PROGRAM PRG_Parada
VAR
	EstoyBloqueandoA: BOOL;
	EstoyBloqueandoV: BOOL;
	EstoyBloqueandoM: BOOL;

	StopBladeA: FB_StopBlade;
	CintaA: 	FB_Cinta;
	
	StopBladeV: FB_StopBlade;
	CintaV: 	FB_Cinta;
	
	StopBladeM: FB_StopBlade;
	CintaM: 	FB_Cinta;
	
	bBloqueoPusherA: BOOL;
	bBloqueoPusherV: BOOL;
	bBloqueoPusherM: BOOL;
END_VAR

(* Mediante este POU se controla el apagado de las líneas en caso de que comiencen a entrar demasiadas piezas en una misma
línea. Mediante su llamada, se impide que haya más de 3 piezas siendo procesadas simultáneamente por cada una de las líneas
del proceso de guardado en cajas. La detención se realiza mediante una llamada a los stopblades que impiden la entrada de
nuevas piezas a los positioner y, a su vez, detiene la cinta de entrada a cada una de las líneas del proceso, impidiendo que
se junten dos piezas seguidas, lo que ocasionaría el colapso total de la línea. *)

// SECCIÓN AZUL
StopBladeA(
	TENERPIEZA:= PRG_Positioner.TengoUnaPiezaA, ESTOYBLOQUEANDO=> EstoyBloqueandoA, 
	STOPBLADE=>GVL_StackBox.bStopBladeA1 );
	
CintaA(
	BLOQUEANDO:= EstoyBloqueandoA, SENSOR:= GVL_StackBox.bRReflectiveSensorA2, 
	CINTA=> GVL_General.sBeltConveyor.bCintaAzul1);

// SECCIÓN VERDE
StopBladeV(
	TENERPIEZA:= PRG_Positioner.TengoUnaPiezaV, ESTOYBLOQUEANDO=> EstoyBloqueandoV, 
	STOPBLADE=>GVL_StackBox.bStopBladeV1 );

CintaV(
	BLOQUEANDO:= EstoyBloqueandoV, SENSOR:= GVL_StackBox.bRReflectiveSensorV2, 
	CINTA=> GVL_General.sBeltConveyor.bCintaVerde1);

// SECCIÓN METAL
StopBladeM(
	TENERPIEZA:= PRG_Positioner.TengoUnaPiezaM, ESTOYBLOQUEANDO=> EstoyBloqueandoM, 
	STOPBLADE=>GVL_StackBox.bStopBladeM1 );

CintaM(
	BLOQUEANDO:= EstoyBloqueandoM, SENSOR:= GVL_StackBox.bRReflectiveSensorM2, 
	CINTA=> GVL_General.sBeltConveyor.bCintaMetal1);


// CONTROL DE ENTRADA	

(* Se tiene en cuenta el llenado de una línea. En caso de que una línea no pueda continuar abarcando
la entrada de piezas, se impide la activación del pusher correspondiente. (Se puede hacer en un FB, no
está hecho así porque me estoy muriendo *)

IF (
	PRG_Positioner.TengoUnaPiezaA AND PRG_PickAndPlace.RobotSeMueveA 
		AND EstoyBloqueandoA AND NOT GVL_General.sBeltConveyor.bCintaAzul1 ) 
THEN
	bBloqueoPusherA := TRUE;
ELSE
	bBloqueoPusherA := FALSE;
END_IF

IF (
	PRG_Positioner.TengoUnaPiezaV AND PRG_PickAndPlace.RobotSeMueveV 
		AND EstoyBloqueandoV AND NOT GVL_General.sBeltConveyor.bCintaVerde1 ) 
THEN
	bBloqueoPusherV := TRUE;
ELSE
	bBloqueoPusherV := FALSE;
END_IF	

IF (
	PRG_Positioner.TengoUnaPiezaM AND PRG_PickAndPlace.RobotSeMueveM 
		AND EstoyBloqueandoM AND NOT GVL_General.sBeltConveyor.bCintaMetal1) 
THEN
	bBloqueoPusherM := TRUE;
ELSE
	bBloqueoPusherM := FALSE;
END_IF

END_PROGRAM

(* stored: Version 1.1.0.1, ProductVersion 3.1.4024.12
   POU PRG_Parada: Id {4562e21a-788d-46be-8a5e-d2163f8820b6}, SpecialFunc None *)
